(* PLC project op_alarms, Dassault Systèmes ControlBuild 2024x *)
(* stored: creationDateTime 2023-10-03T11:13:51-01:00 *)

PROGRAM tni_train.op_alarms
  VAR_OUTPUT
    AlarmD1L : BOOL := false;
    AlarmD2L : BOOL := false;
    AlarmD3L : BOOL := false;
    AlarmD1R : BOOL := false;
    AlarmD2R : BOOL := false;
    AlarmD3R : BOOL := false;
  END_VAR

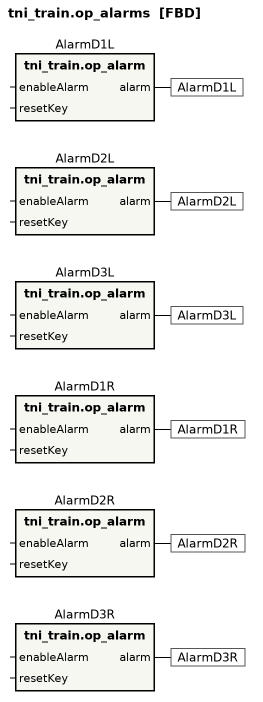
(* FBD diagram, written out as Structured Text *)
AlarmD1L();
AlarmD1L := AlarmD1L.alarm;
AlarmD2L();
AlarmD2L := AlarmD2L.alarm;
AlarmD3L();
AlarmD3L := AlarmD3L.alarm;
AlarmD1R();
AlarmD1R := AlarmD1R.alarm;
AlarmD2R();
AlarmD2R := AlarmD2R.alarm;
AlarmD3R();
AlarmD3R := AlarmD3R.alarm;
END_PROGRAM
